TYPE U_Arrays2DimInOne :

UNION
	nData	: ARRAY[1..nMaxReadDataArray_2Dim] OF BYTE;
	bBool	: ARRAY[1..nArrayTestLength_2DimX, 1..nArrayTestLength_2DimY] OF BOOL;
	bByte	: ARRAY[1..nArrayTestLength_2DimX, 1..nArrayTestLength_2DimY] OF BYTE;
	nInt	: ARRAY[1..nArrayTestLength_2DimX, 1..nArrayTestLength_2DimY] OF INT;
	nUdint	: ARRAY[1..nArrayTestLength_2DimX, 1..nArrayTestLength_2DimY] OF UDINT;
	nReal	: ARRAY[1..nArrayTestLength_2DimX, 1..nArrayTestLength_2DimY] OF REAL;
	nLReal	: ARRAY[1..nArrayTestLength_2DimX, 1..nArrayTestLength_2DimY] OF LREAL;
	sString	: ARRAY[1..nArrayTestLength_2DimX, 1..nArrayTestLength_2DimY] OF STRING(80);
	wLword	: ARRAY[1..nArrayTestLength_2DimX, 1..nArrayTestLength_2DimY] OF LWORD;
	dDate	: ARRAY[1..nArrayTestLength_2DimX, 1..nArrayTestLength_2DimY] OF DT;
END_UNION

END_TYPE

(* stored: Version 1.1.0.1, ProductVersion 3.1.0.24
   DUT U_Arrays2DimInOne: Id {ed3889f0-2727-4978-a1fa-714db5b6d4fe} *)
